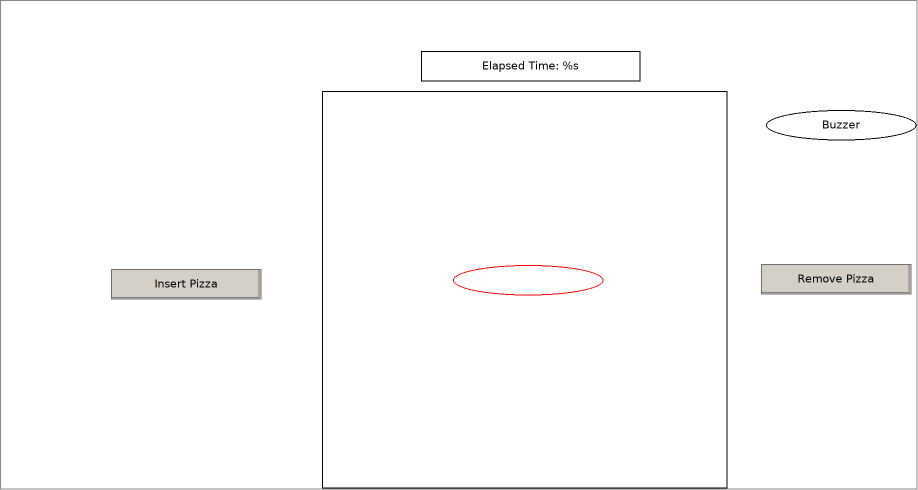
VISUALIZATION Visualization_1  // 918x490
    Rectangle (322,91 405x397)
    Button (111,269 150x30), "Insert Pizza"
        OnMouseDown: execute { MAIN.bPizzaInOven := TRUE; }
    Button (761,264 150x30), "Remove Pizza"
        OnMouseDown: execute { MAIN.bPizzaInOven := FALSE; }
    Ellipse (453,265 150x30), invisible if: NOT MAIN.bPizzaInOven
    Rectangle (421,51 219x30), "Elapsed Time: %s", text variable: MAIN.fbMyTimer.ET
    Ellipse (766,110 150x30), "Buzzer", colour toggle: MAIN.bBuzzer
END_VISUALIZATION

(* stored: Version 1.1.0.1, ProductVersion 3.1.4019.2
   Visu Visualization_1: Id {2a13d671-806b-4046-a974-7bc98291b730} *)
